(* IEC 61131-3 sources: inproshop/TEAM_V2.0-demo_exported/1.Function/FB/Gear(电子齿轮控制), 5 files *)

(* ---- Str_Gear.st ---- *)
TYPE Str_Gear :
STRUCT
	Cmd:Str_GearCmd;//控制
	Parm:Str_GearParm;//参数
	Status:Str_GearStatus;//状态
END_STRUCT
END_TYPE

(* ---- Str_GearCmd.st ---- *)
TYPE Str_GearCmd :
STRUCT
	GearIn:BOOL;//耦合
	GearOut:BOOL;//解耦
END_STRUCT
END_TYPE

(* ---- Str_GearParm.st ---- *)
TYPE Str_GearParm :
STRUCT
	IC_Home:BOOL;//回原互锁条件
	IC_ABS:BOOL;//定位互锁条件
	IC_JOG:BOOL;//点动互锁条件
	_ABS:ARRAY[0..49] OF Str_AxisParmControl;
	_INC:ARRAY[0..49] OF Str_AxisParmControl;
	ManuPosition:REAL;//手动定位点位
	ManuVelocity:REAL;//手动定位速度
	VelModeVelocity:REAL;//速度模式定位速度
	Comment:WSTRING(40);//轴名称
END_STRUCT
END_TYPE

(* ---- Str_GearStatus.st ---- *)
TYPE Str_GearStatus :
STRUCT
	InGear:BOOL;//从轴已耦合
	Error:BOOL;//错误
	ErrorID:WORD;//错误代码
END_STRUCT
END_TYPE

(* ---- FB_Gear.st ---- *)
FUNCTION_BLOCK FB_Gear
VAR_IN_OUT
	ioMaster:AXIS_REF_SM3;//主轴
	ioSlave:AXIS_REF_SM3;//从轴
	ioGear:Str_Gear;//控制
END_VAR
VAR_INPUT
	iEstop:BOOL;//急停信号
	iRatioNumerator:DINT := 1;//齿轮比分子
	iRatioDenominator:UDINT := 1;//齿轮比分母
END_VAR
VAR_OUTPUT
END_VAR
VAR
	MC_GearIn_0: MC_GearIn;
	MC_GearOut_0: MC_GearOut;
	MC_Stop_0: MC_Stop;
END_VAR

//主轴未使能，轴报错，轴回原中 不可以耦合
IF ioMaster.nAxisState <> 0 AND ioSlave.nAxisState <> 0 AND ioMaster.nAxisState <> 1 AND ioMaster.nAxisState<>7 THEN
	ioGear.Cmd.GearIn:=FALSE;
END_IF

//从轴异常 控制解耦
IF ioSlave.nAxisState = 1 THEN
	ioGear.Cmd.GearOut:=TRUE;
END_IF
//解耦
IF ioGear.Cmd.GearOut THEN
	MC_GearIn_0.Execute:=FALSE;
END_IF

//耦合实例化
MC_GearIn_0(
	Master:= ioMaster,
	Slave:= ioSlave,
	Execute:= MC_GearIn_0.Execute ,
	RatioNumerator:= iRatioNumerator,
	RatioDenominator:= iRatioDenominator,
	Acceleration:= ,
	Deceleration:= ,
	Jerk:= ,
	BufferMode:= ,
	InGear=> ioGear.Status.InGear,
	Busy=> ,
	Active=> ,
	CommandAborted=> ,
	Error=> ,
	ErrorID=> );

//解耦实例化
MC_GearOut_0(
	Slave:= ioSlave,
	Execute:= ioGear.Cmd.GearOut,
	Done=> ,
	Busy=> ,
	Error=> ,
	ErrorID=> );

(*********解耦后触发轴停止，防止从轴继续运行*************)
//停止轴实例化
MC_Stop_0(
	Axis:= ioSlave,
	Execute:= MC_GearOut_0.Done,
	Deceleration:= ,
	Jerk:= ,
	Done=> ,
	Busy=> ,
	Error=> ,
	ErrorID=> );
